// TIA Portal V20 export
// export: Created 2026-07-10T11:12:34.3299646Z, ExportSetting WithDefaults, DisplayName Totally Integrated Automation Portal, DisplayVersion V20, DisplayName TIA Portal Openness, DisplayVersion V20, DisplayName TIA Portal Version Control Interface, DisplayVersion V20, DisplayName STEP 7 Professional, DisplayVersion V20, DisplayName STEP 7 Safety, DisplayVersion V20, DisplayName WinCC Basic/Comfort/Advanced, DisplayVersion V20, DisplayName WinCC Unified, DisplayVersion V20
FUNCTION_BLOCK "TankRegistrator"   // FB24, SCL
{ S7_Optimized_Access := 'TRUE' }
VERSION : 0.1
// stored: AutoNumber true, IsIECCheckEnabled false, IsRetainMemResEnabled false, MemoryReserve 100, SetENOAutomatically false, UDAEnableTagReadback false
   VAR_INPUT
      CurrentConsumedFeed1 : Real;
      CurrentConsumedFeed2 : Real;
      CurrentLoadedFeed1 : Real;
      CurrentLoadedFeed2 : Real;
      DayTour : Int;
      CalendarDay : UInt;
      CalendarMonth : UInt;
   END_VAR
   VAR_OUTPUT
      ResetCounters : Bool;
   END_VAR
   VAR_IN_OUT
      ref_RetainData : "WeightRetainData";
   END_VAR
   VAR
      i : Int;
   END_VAR
   VAR CONSTANT
      c_ARRAY_SIZE : Int := 30;
   END_VAR
BEGIN

   IF #ref_RetainData.PreviousDayTour <> #DayTour THEN
       FOR #i := 0 TO (#c_ARRAY_SIZE - 2) DO
           #ref_RetainData.ArrayConsumedFeed1[c_ARRAY_SIZE - #i] := #ref_RetainData.ArrayConsumedFeed1[c_ARRAY_SIZE - #i - 1];
           #ref_RetainData.ArrayLoadedFeed1[c_ARRAY_SIZE - #i] := #ref_RetainData.ArrayLoadedFeed1[c_ARRAY_SIZE - #i - 1];
           #ref_RetainData.ArrayConsumedFeed2[c_ARRAY_SIZE - #i] := #ref_RetainData.ArrayConsumedFeed2[c_ARRAY_SIZE - #i - 1];
           #ref_RetainData.ArrayLoadedFeed2[c_ARRAY_SIZE - #i] := #ref_RetainData.ArrayLoadedFeed2[c_ARRAY_SIZE - #i - 1];
           #ref_RetainData.ArrayDayTour[c_ARRAY_SIZE - #i] := #ref_RetainData.ArrayDayTour[c_ARRAY_SIZE - #i - 1];
           #ref_RetainData.ArrayCalendarDay[c_ARRAY_SIZE - #i] := #ref_RetainData.ArrayCalendarDay[c_ARRAY_SIZE - #i - 1];
           #ref_RetainData.ArrayCalendarMonth[c_ARRAY_SIZE - #i] := #ref_RetainData.ArrayCalendarMonth[c_ARRAY_SIZE - #i - 1];
       END_FOR;
       #ref_RetainData.PreviousDayTour := #DayTour;
       #ResetCounters := TRUE;
   ELSE
       #ResetCounters := FALSE;
   END_IF;

       #ref_RetainData.ArrayConsumedFeed1[1] := #CurrentConsumedFeed1;
       #ref_RetainData.ArrayLoadedFeed1[1] := #CurrentLoadedFeed1;
       #ref_RetainData.ArrayConsumedFeed2[1] := #CurrentConsumedFeed2;
       #ref_RetainData.ArrayLoadedFeed2[1] := #CurrentLoadedFeed2;
       #ref_RetainData.ArrayDayTour[1] := #DayTour;
       #ref_RetainData.ArrayCalendarDay[1] := #CalendarDay;
       #ref_RetainData.ArrayCalendarMonth[1] := #CalendarMonth;
END_FUNCTION_BLOCK
